// Mitsubishi GX Works2 project: 시퀀스 무한 반복 예제   PLC: Q03UDV

PROGRAM MAIN
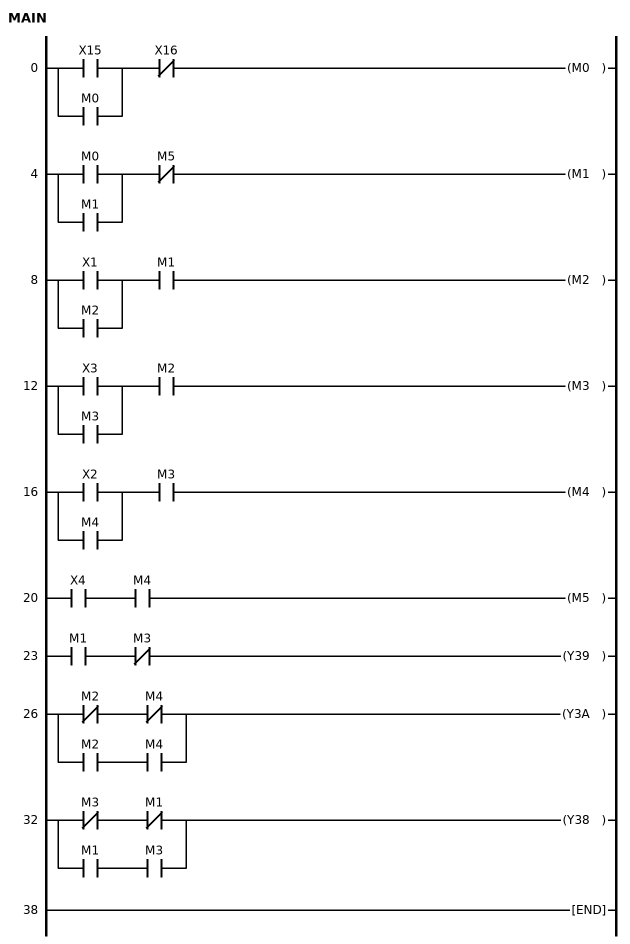
0     LD      X15
      OR      M0
      ANI     X16
      OUT     M0
4     LD      M0
      OR      M1
      ANI     M5
      OUT     M1
8     LD      X1
      OR      M2
      AND     M1
      OUT     M2
12    LD      X3
      OR      M3
      AND     M2
      OUT     M3
16    LD      X2
      OR      M4
      AND     M3
      OUT     M4
20    LD      X4
      AND     M4
      OUT     M5
23    LD      M1
      ANI     M3
      OUT     Y39
26    LDI     M2
      ANI     M4
      LD      M2
      AND     M4
      ORB
      OUT     Y3A
32    LDI     M3
      ANI     M1
      LD      M1
      AND     M3
      ORB
      OUT     Y38
38    END
END_PROGRAM
